(* PLC project PLC, Beckhoff Automation GmbH TwinCAT PLC Control 3.5.13.20 *)
(* stored: creationDateTime 2021-09-02T10:22:54.9959735, modificationDateTime 2021-09-02T10:22:54.9959735 *)

(*-----------------------------------------版本信息-----------------------------------------
第一版本：		V1.0.0
功能说明：		边缘触发功能块集合
开发者：		Long.Yun
开发时间：		2021.09.02

变更版本：
版本			变更者		变更时间		变更说明
------------------------------------------------------------------------------------------*)
{attribute 'hide_all_locals'}
FUNCTION_BLOCK BFB_Trigger
VAR_INPUT
	//触发位
	bIn			:BOOL;
END_VAR

VAR_OUTPUT
	//边沿交替输出
	bTrig		:BOOL;
	//上升沿输出
	bRiseTrig	:BOOL;
	//下降沿输出
	bFallTrig	:BOOL;
END_VAR

VAR
	fbTrigR		:R_TRIG;
	fbTrigF		:F_TRIG;
END_VAR

            fbTrigR(CLK := bIn, Q =>bRiseTrig);

fbTrigF(CLK := bIn, Q => bFallTrig);

bTrig := bRiseTrig OR bFallTrig;
          
END_FUNCTION_BLOCK
